// TIA Portal V21 export
VAR_GLOBAL   // PLC tag table "InputAnalogici"
   Tag_1 AT %IW200 : Word;   // Commento / Comment / Comentario
END_VAR
